{attribute addProperty BoxType "EK1122-0000-0018"}
{attribute addProperty Id "Beckhoff_EK18xxsub_EK1100EK1100_179A0949162A_0001_EK1814_0000_0016EK1814_97B4DD118210.25A_0002_EK1814_0000_0017EK1814_97B4DD118210.25A_0003_EK1814_0000_0018EK1814_97B4DD118210.25A_0004_EK1814_0000_0019EK1814_97B4DD118210.25A_0005_EK1818_0000_0016EK1818_5F755A8411414.25A_0006_EK1818_0000_0017EK1818_5F755A8411414.25A_0007_EK1818_0000_0018EK1818_5F755A8411414.25A_0008_EK1828_0000_0016EK1828_A5978B6311414.25A_0009_EK1828_0000_0017EK1828_A5978B6311414.25A_0010_EK1828_0000_0018EK1828_A5978B6311414.25A_0011_EK1828_0010_0016EK1828_A854BE6D8110.125A_0012_EK1828_0010_0017EK1828_A854BE6D8110.125A_0013_EK1828_0010_0018EK1828_A854BE6D8110.125"}
{attribute addProperty CRC "1186666968"}
{attribute addProperty SizeInBites "1271"}
{attribute addProperty SizeInBytes "158.875"}
TYPE Beckhoff_EK18xxEK1122_46BB19D8 EXTENDS EK1122_179A0949 :
STRUCT
	{attribute addProperty Name "Beckhoff_EK18xxsub_EK1100"}
	Beckhoff_EK18xxsub_EK1100 : EK1100_179A0949;
	{attribute addProperty Name "A_0001_EK1814_0000_0016"}
	A_0001_EK1814_0000_0016 : EK1814_97B4DD11;
	{attribute addProperty Name "A_0002_EK1814_0000_0017"}
	A_0002_EK1814_0000_0017 : EK1814_97B4DD11;
	{attribute addProperty Name "A_0003_EK1814_0000_0018"}
	A_0003_EK1814_0000_0018 : EK1814_97B4DD11;
	{attribute addProperty Name "A_0004_EK1814_0000_0019"}
	A_0004_EK1814_0000_0019 : EK1814_97B4DD11;
	{attribute addProperty Name "A_0005_EK1818_0000_0016"}
	A_0005_EK1818_0000_0016 : EK1818_5F755A84;
	{attribute addProperty Name "A_0006_EK1818_0000_0017"}
	A_0006_EK1818_0000_0017 : EK1818_5F755A84;
	{attribute addProperty Name "A_0007_EK1818_0000_0018"}
	A_0007_EK1818_0000_0018 : EK1818_5F755A84;
	{attribute addProperty Name "A_0008_EK1828_0000_0016"}
	A_0008_EK1828_0000_0016 : EK1828_A5978B63;
	{attribute addProperty Name "A_0009_EK1828_0000_0017"}
	A_0009_EK1828_0000_0017 : EK1828_A5978B63;
	{attribute addProperty Name "A_0010_EK1828_0000_0018"}
	A_0010_EK1828_0000_0018 : EK1828_A5978B63;
	{attribute addProperty Name "A_0011_EK1828_0010_0016"}
	A_0011_EK1828_0010_0016 : EK1828_A854BE6D;
	{attribute addProperty Name "A_0012_EK1828_0010_0017"}
	A_0012_EK1828_0010_0017 : EK1828_A854BE6D;
	{attribute addProperty Name "A_0013_EK1828_0010_0018"}
	A_0013_EK1828_0010_0018 : EK1828_A854BE6D;
END_STRUCT
END_TYPE

(* stored: Version 1.2.0.0, ProductVersion 3.1.4024.9
   DUT Beckhoff_EK18xxEK1122_46BB19D8: Id {f1edbab1-08aa-4f03-a837-9a1223981948} *)
